  gc_ErrTranslation_fr_Text612 : WSTRING(60) := " [PIN_180 ]: EvPropGenerator -  Deviation of current control";
  gc_ErrTranslation_fr_Text613 : WSTRING(77) := " [PIN_180 ]: EvPropGenerator -  Internal error ( software or hardware error )";
  gc_ErrTranslation_fr_Text614 : WSTRING(65) := " [PIN_189 ]: EvServiceBrakeAxleOscillant -  Internal Driver Error";
  gc_ErrTranslation_fr_Text615 : WSTRING(13) := "Unknown error";
  gc_ErrTranslation_fr_Text616 : WSTRING(32) := "Short to Power has been detected";
  gc_ErrTranslation_fr_Text617 : WSTRING(33) := "Short to Ground has been detected";
  gc_ErrTranslation_fr_Text618 : WSTRING(15) := "Wrong Parameter";
  gc_ErrTranslation_fr_Text619 : WSTRING(13) := "Unknown error";
  gc_ErrTranslation_fr_Text620 : WSTRING(32) := "Short to Power has been detected";
  gc_ErrTranslation_fr_Text621 : WSTRING(33) := "Short to Ground has been detected";
  gc_ErrTranslation_fr_Text622 : WSTRING(15) := "Wrong Parameter";
  gc_ErrTranslation_fr_Text623 : WSTRING(13) := "Unknown error";
  gc_ErrTranslation_fr_Text624 : WSTRING(71) := " [PIN_193 ]: EvUpAxleOscillant -  HS OpenLoad / Short To Power external";
  gc_ErrTranslation_fr_Text625 : WSTRING(60) := " [PIN_193 ]: EvUpAxleOscillant -  HS Short To Power internal";
  gc_ErrTranslation_fr_Text626 : WSTRING(52) := " [PIN_193 ]: EvUpAxleOscillant -  HS Short To Ground";
  gc_ErrTranslation_fr_Text627 : WSTRING(55) := " [PIN_193 ]: EvUpAxleOscillant -  Internal Driver Error";
  gc_ErrTranslation_fr_Text628 : WSTRING(37) := "HS OpenLoad / Short To Power external";
  gc_ErrTranslation_fr_Text629 : WSTRING(26) := "HS Short To Power internal";
  gc_ErrTranslation_fr_Text630 : WSTRING(18) := "HS Short To Ground";
  gc_ErrTranslation_fr_Text631 : WSTRING(21) := "Internal Driver Error";
  gc_ErrTranslation_fr_Text632 : WSTRING(37) := "HS OpenLoad / Short To Power external";
  gc_ErrTranslation_fr_Text633 : WSTRING(26) := "HS Short To Power internal";
  gc_ErrTranslation_fr_Text634 : WSTRING(18) := "HS Short To Ground";
  gc_ErrTranslation_fr_Text635 : WSTRING(21) := "Internal Driver Error";
  gc_ErrTranslation_fr_Text636 : WSTRING(52) := "An input signal is too low / Short circuit to ground";
  gc_ErrTranslation_fr_Text637 : WSTRING(52) := "An input signal is too high / Short circuit to power";
  gc_ErrTranslation_fr_Text638 : WSTRING(37) := "An input signal is out of valid range";
  gc_ErrTranslation_fr_Text639 : WSTRING(39) := "Warning: a block has limited parameters";
  gc_ErrTranslation_fr_Text640 : WSTRING(23) := "An initialization error";
  gc_ErrTranslation_fr_Text641 : WSTRING(52) := "An input signal is too low / Short circuit to ground";
  gc_ErrTranslation_fr_Text642 : WSTRING(52) := "An input signal is too high / Short circuit to power";
  gc_ErrTranslation_fr_Text643 : WSTRING(37) := "An input signal is out of valid range";
  gc_ErrTranslation_fr_Text644 : WSTRING(39) := "Warning: a block has limited parameters";
  gc_ErrTranslation_fr_Text645 : WSTRING(23) := "An initialization error";
  gc_ErrTranslation_fr_Text646 : WSTRING(66) := " [PIN_196 ]: EvUpAxleFixe -  HS OpenLoad / Short To Power external";
  gc_ErrTranslation_fr_Text647 : WSTRING(55) := " [PIN_196 ]: EvUpAxleFixe -  HS Short To Power internal";
  gc_ErrTranslation_fr_Text648 : WSTRING(47) := " [PIN_196 ]: EvUpAxleFixe -  HS Short To Ground";
  gc_ErrTranslation_fr_Text649 : WSTRING(50) := " [PIN_196 ]: EvUpAxleFixe -  Internal Driver Error";
  gc_ErrTranslation_fr_Text650 : WSTRING(73) := " [PIN_169 ]: EvDownAxleOscillant -  HS OpenLoad / Short To Power external";
  gc_ErrTranslation_fr_Text651 : WSTRING(62) := " [PIN_149 ]: BlueFire -  HS OpenLoad / Short To Power external";
  gc_ErrTranslation_fr_Text652 : WSTRING(51) := " [PIN_149 ]: BlueFire -  HS Short To Power internal";
  gc_ErrTranslation_fr_Text653 : WSTRING(43) := " [PIN_149 ]: BlueFire -  HS Short To Ground";
  gc_ErrTranslation_fr_Text654 : WSTRING(46) := " [PIN_149 ]: BlueFire -  Internal Driver Error";
  gc_ErrTranslation_fr_Text655 : WSTRING(73) := " [PIN_173 ]: OrangeFlashingLight -  HS OpenLoad / Short To Power external";
  gc_ErrTranslation_fr_Text656 : WSTRING(62) := " [PIN_173 ]: OrangeFlashingLight -  HS Short To Power internal";
  gc_ErrTranslation_fr_Text657 : WSTRING(54) := " [PIN_173 ]: OrangeFlashingLight -  HS Short To Ground";
  gc_ErrTranslation_fr_Text658 : WSTRING(57) := " [PIN_173 ]: OrangeFlashingLight -  Internal Driver Error";
  gc_ErrTranslation_fr_Text659 : WSTRING(62) := " [PIN_169 ]: EvDownAxleOscillant -  HS Short To Power internal";
  gc_ErrTranslation_fr_Text660 : WSTRING(54) := " [PIN_169 ]: EvDownAxleOscillant -  HS Short To Ground";
  gc_ErrTranslation_fr_Text661 : WSTRING(57) := " [PIN_169 ]: EvDownAxleOscillant -  Internal Driver Error";
  gc_ErrTranslation_fr_Text662 : WSTRING(68) := " [PIN_172 ]: EvDownAxleFixe -  HS OpenLoad / Short To Power external";
  gc_ErrTranslation_fr_Text663 : WSTRING(62) := " [PIN_182 ]: EvBypass -  HS OpenLoad / Short To Power external";
  gc_ErrTranslation_fr_Text664 : WSTRING(51) := " [PIN_182 ]: EvBypass -  HS Short To Power internal";
  gc_ErrTranslation_fr_Text665 : WSTRING(43) := " [PIN_182 ]: EvBypass -  HS Short To Ground";
  gc_ErrTranslation_fr_Text666 : WSTRING(46) := " [PIN_182 ]: EvBypass -  Internal Driver Error";
  gc_ErrTranslation_fr_Text667 : WSTRING(57) := " [PIN_172 ]: EvDownAxleFixe -  HS Short To Power internal";
  gc_ErrTranslation_fr_Text668 : WSTRING(49) := " [PIN_172 ]: EvDownAxleFixe -  HS Short To Ground";
  gc_ErrTranslation_fr_Text669 : WSTRING(52) := " [PIN_172 ]: EvDownAxleFixe -  Internal Driver Error";
  gc_ErrTranslation_fr_Text670 : WSTRING(71) := " [PIN_191 ]: SupplyPvgDeltaArm -  HS OpenLoad / Short To Power external";
  gc_ErrTranslation_fr_Text671 : WSTRING(60) := " [PIN_191 ]: SupplyPvgDeltaArm -  HS Short To Power internal";
  gc_ErrTranslation_fr_Text672 : WSTRING(52) := " [PIN_191 ]: SupplyPvgDeltaArm -  HS Short To Ground";
  gc_ErrTranslation_fr_Text673 : WSTRING(55) := " [PIN_191 ]: SupplyPvgDeltaArm -  Internal Driver Error";
  gc_ErrTranslation_fr_Text674 : WSTRING(70) := " [PIN_167 ]: SupplyPvgBoomArm -  HS OpenLoad / Short To Power external";
  gc_ErrTranslation_fr_Text675 : WSTRING(59) := " [PIN_167 ]: SupplyPvgBoomArm -  HS Short To Power internal";
  gc_ErrTranslation_fr_Text676 : WSTRING(51) := " [PIN_167 ]: SupplyPvgBoomArm -  HS Short To Ground";
  gc_ErrTranslation_fr_Text677 : WSTRING(54) := " [PIN_167 ]: SupplyPvgBoomArm -  Internal Driver Error";
  gc_ErrTranslation_fr_Text678 : WSTRING(75) := " [PIN_194 ]: SupplyPvgTelescopeArm -  HS OpenLoad / Short To Power external";
  gc_ErrTranslation_fr_Text679 : WSTRING(64) := " [PIN_194 ]: SupplyPvgTelescopeArm -  HS Short To Power internal";
  gc_ErrTranslation_fr_Text680 : WSTRING(56) := " [PIN_194 ]: SupplyPvgTelescopeArm -  HS Short To Ground";
  gc_ErrTranslation_fr_Text681 : WSTRING(59) := " [PIN_194 ]: SupplyPvgTelescopeArm -  Internal Driver Error";
  gc_ErrTranslation_fr_Text682 : WSTRING(72) := " [PIN_170 ]: SupplyPvgPropEvTOR -  HS OpenLoad / Short To Power external";
  gc_ErrTranslation_fr_Text683 : WSTRING(61) := " [PIN_170 ]: SupplyPvgPropEvTOR -  HS Short To Power internal";
  gc_ErrTranslation_fr_Text684 : WSTRING(53) := " [PIN_170 ]: SupplyPvgPropEvTOR -  HS Short To Ground";
  gc_ErrTranslation_fr_Text685 : WSTRING(56) := " [PIN_170 ]: SupplyPvgPropEvTOR -  Internal Driver Error";
  gc_ErrTranslation_fr_Text686 : WSTRING(83) := " [PIN_110 ]: RailHookSensor -  An input signal is too high / Short circuit to power";
  gc_ErrTranslation_fr_Text687 : WSTRING(68) := " [PIN_110 ]: RailHookSensor -  An input signal is out of valid range";
  gc_ErrTranslation_fr_Text688 : WSTRING(70) := " [PIN_110 ]: RailHookSensor -  Warning: a block has limited parameters";
  gc_ErrTranslation_fr_Text689 : WSTRING(54) := " [PIN_110 ]: RailHookSensor -  An initialization error";
  gc_ErrTranslation_fr_Text690 : WSTRING(88) := " [PIN_134 ]: InductiveRailSensor -  An input signal is too low / Short circuit to ground";
  gc_ErrTranslation_fr_Text691 : WSTRING(88) := " [PIN_134 ]: InductiveRailSensor -  An input signal is too high / Short circuit to power";
  gc_ErrTranslation_fr_Text692 : WSTRING(73) := " [PIN_134 ]: InductiveRailSensor -  An input signal is out of valid range";
  gc_ErrTranslation_fr_Text693 : WSTRING(75) := " [PIN_134 ]: InductiveRailSensor -  Warning: a block has limited parameters";
  gc_ErrTranslation_fr_Text694 : WSTRING(59) := " [PIN_134 ]: InductiveRailSensor -  An initialization error";
  gc_ErrTranslation_fr_Text695 : WSTRING(83) := " [PIN_111 ]: CenteredTurret -  An input signal is too low / Short circuit to ground";
  gc_ErrTranslation_fr_Text696 : WSTRING(83) := " [PIN_111 ]: CenteredTurret -  An input signal is too high / Short circuit to power";
  gc_ErrTranslation_fr_Text697 : WSTRING(68) := " [PIN_111 ]: CenteredTurret -  An input signal is out of valid range";
  gc_ErrTranslation_fr_Text698 : WSTRING(70) := " [PIN_111 ]: CenteredTurret -  Warning: a block has limited parameters";
  gc_ErrTranslation_fr_Text699 : WSTRING(54) := " [PIN_111 ]: CenteredTurret -  An initialization error";
  gc_ErrTranslation_fr_Text700 : WSTRING(85) := " [PIN_135 ]: WorkKeyTrackSide -  An input signal is too low / Short circuit to ground";
  gc_ErrTranslation_fr_Text701 : WSTRING(85) := " [PIN_135 ]: WorkKeyTrackSide -  An input signal is too high / Short circuit to power";
  gc_ErrTranslation_fr_Text702 : WSTRING(70) := " [PIN_135 ]: WorkKeyTrackSide -  An input signal is out of valid range";
  gc_ErrTranslation_fr_Text703 : WSTRING(72) := " [PIN_135 ]: WorkKeyTrackSide -  Warning: a block has limited parameters";
  gc_ErrTranslation_fr_Text704 : WSTRING(56) := " [PIN_135 ]: WorkKeyTrackSide -  An initialization error";
  gc_ErrTranslation_fr_Text705 : WSTRING(85) := " [PIN_136 ]: WorkKeyBilateral -  An input signal is too low / Short circuit to ground";
  gc_ErrTranslation_fr_Text706 : WSTRING(85) := " [PIN_136 ]: WorkKeyBilateral -  An input signal is too high / Short circuit to power";
  gc_ErrTranslation_fr_Text707 : WSTRING(70) := " [PIN_136 ]: WorkKeyBilateral -  An input signal is out of valid range";
  gc_ErrTranslation_fr_Text708 : WSTRING(72) := " [PIN_136 ]: WorkKeyBilateral -  Warning: a block has limited parameters";
  gc_ErrTranslation_fr_Text709 : WSTRING(56) := " [PIN_136 ]: WorkKeyBilateral -  An initialization error";
  gc_ErrTranslation_fr_Text710 : WSTRING(83) := " [PIN_113 ]: WorkKeyCentred -  An input signal is too low / Short circuit to ground";
  gc_ErrTranslation_fr_Text711 : WSTRING(83) := " [PIN_113 ]: WorkKeyCentred -  An input signal is too high / Short circuit to power";
  gc_ErrTranslation_fr_Text712 : WSTRING(68) := " [PIN_113 ]: WorkKeyCentred -  An input signal is out of valid range";
  gc_ErrTranslation_fr_Text713 : WSTRING(70) := " [PIN_113 ]: WorkKeyCentred -  Warning: a block has limited parameters";
  gc_ErrTranslation_fr_Text714 : WSTRING(54) := " [PIN_113 ]: WorkKeyCentred -  An initialization error";
  gc_ErrTranslation_fr_Text715 : WSTRING(92) := " [PIN_137 ]: AbutmentTurretTrackSide -  An input signal is too low / Short circuit to ground";
  gc_ErrTranslation_fr_Text716 : WSTRING(92) := " [PIN_137 ]: AbutmentTurretTrackSide -  An input signal is too high / Short circuit to power";
  gc_ErrTranslation_fr_Text717 : WSTRING(77) := " [PIN_137 ]: AbutmentTurretTrackSide -  An input signal is out of valid range";
  gc_ErrTranslation_fr_Text718 : WSTRING(79) := " [PIN_137 ]: AbutmentTurretTrackSide -  Warning: a block has limited parameters";
  gc_ErrTranslation_fr_Text719 : WSTRING(63) := " [PIN_137 ]: AbutmentTurretTrackSide -  An initialization error";
  gc_ErrTranslation_fr_Text720 : WSTRING(94) := " [PIN_138 ]: AbutmentTurretCentredSide -  An input signal is too low / Short circuit to ground";
  gc_ErrTranslation_fr_Text721 : WSTRING(94) := " [PIN_138 ]: AbutmentTurretCentredSide -  An input signal is too high / Short circuit to power";
  gc_ErrTranslation_fr_Text722 : WSTRING(79) := " [PIN_138 ]: AbutmentTurretCentredSide -  An input signal is out of valid range";
  gc_ErrTranslation_fr_Text723 : WSTRING(81) := " [PIN_138 ]: AbutmentTurretCentredSide -  Warning: a block has limited parameters";
  gc_ErrTranslation_fr_Text724 : WSTRING(65) := " [PIN_138 ]: AbutmentTurretCentredSide -  An initialization error";
  gc_ErrTranslation_fr_Text725 : WSTRING(96) := " [PIN_139 ]: OscillantAxleSpeedSensorDir -  An input signal is too low / Short circuit to ground";
  gc_ErrTranslation_fr_Text726 : WSTRING(96) := " [PIN_139 ]: OscillantAxleSpeedSensorDir -  An input signal is too high / Short circuit to power";
  gc_ErrTranslation_fr_Text727 : WSTRING(81) := " [PIN_139 ]: OscillantAxleSpeedSensorDir -  An input signal is out of valid range";
  gc_ErrTranslation_fr_Text728 : WSTRING(83) := " [PIN_139 ]: OscillantAxleSpeedSensorDir -  Warning: a block has limited parameters";
  gc_ErrTranslation_fr_Text729 : WSTRING(67) := " [PIN_139 ]: OscillantAxleSpeedSensorDir -  An initialization error";
  gc_ErrTranslation_fr_Text730 : WSTRING(91) := " [PIN_140 ]: FixeAxleSpeedSensorDir -  An input signal is too low / Short circuit to ground";
  gc_ErrTranslation_fr_Text731 : WSTRING(91) := " [PIN_140 ]: FixeAxleSpeedSensorDir -  An input signal is too high / Short circuit to power";
  gc_ErrTranslation_fr_Text732 : WSTRING(76) := " [PIN_140 ]: FixeAxleSpeedSensorDir -  An input signal is out of valid range";
  gc_ErrTranslation_fr_Text733 : WSTRING(78) := " [PIN_140 ]: FixeAxleSpeedSensorDir -  Warning: a block has limited parameters";
  gc_ErrTranslation_fr_Text734 : WSTRING(62) := " [PIN_140 ]: FixeAxleSpeedSensorDir -  An initialization error";
  gc_ErrTranslation_fr_Text735 : WSTRING(81) := " [PIN_117 ]: TrailerGache -  An input signal is too low / Short circuit to ground";
  gc_ErrTranslation_fr_Text736 : WSTRING(81) := " [PIN_117 ]: TrailerGache -  An input signal is too high / Short circuit to power";
  gc_ErrTranslation_fr_Text737 : WSTRING(66) := " [PIN_117 ]: TrailerGache -  An input signal is out of valid range";
  gc_ErrTranslation_fr_Text738 : WSTRING(68) := " [PIN_117 ]: TrailerGache -  Warning: a block has limited parameters";
  gc_ErrTranslation_fr_Text739 : WSTRING(52) := " [PIN_117 ]: TrailerGache -  An initialization error";
  gc_ErrTranslation_fr_Text740 : WSTRING(94) := " [PIN_141 ]: MeasuringMastSensorFolded -  An input signal is too low / Short circuit to ground";
  gc_ErrTranslation_fr_Text741 : WSTRING(94) := " [PIN_141 ]: MeasuringMastSensorFolded -  An input signal is too high / Short circuit to power";
  gc_ErrTranslation_fr_Text742 : WSTRING(79) := " [PIN_141 ]: MeasuringMastSensorFolded -  An input signal is out of valid range";
  gc_ErrTranslation_fr_Text743 : WSTRING(81) := " [PIN_141 ]: MeasuringMastSensorFolded -  Warning: a block has limited parameters";
  gc_ErrTranslation_fr_Text744 : WSTRING(65) := " [PIN_141 ]: MeasuringMastSensorFolded -  An initialization error";
  gc_ErrTranslation_fr_Text745 : WSTRING(80) := " [PIN_124 ]: Aru1Contact -  An input signal is too low / Short circuit to ground";
  gc_ErrTranslation_fr_Text746 : WSTRING(80) := " [PIN_124 ]: Aru1Contact -  An input signal is too high / Short circuit to power";
  gc_ErrTranslation_fr_Text747 : WSTRING(65) := " [PIN_124 ]: Aru1Contact -  An input signal is out of valid range";
  gc_ErrTranslation_fr_Text748 : WSTRING(67) := " [PIN_124 ]: Aru1Contact -  Warning: a block has limited parameters";
  gc_ErrTranslation_fr_Text749 : WSTRING(54) := " [PIN_101 ]: EvForwardPump -  Open load / open circuit";
  gc_ErrTranslation_fr_Text750 : WSTRING(69) := " [PIN_101 ]: EvForwardPump -  Short circuit to power supply / battery";
  gc_ErrTranslation_fr_Text751 : WSTRING(53) := " [PIN_101 ]: EvForwardPump -  Short circuit to ground";
  gc_ErrTranslation_fr_Text752 : WSTRING(58) := " [PIN_101 ]: EvForwardPump -  Deviation of current control";
  gc_ErrTranslation_fr_Text753 : WSTRING(75) := " [PIN_101 ]: EvForwardPump -  Internal error ( software or hardware error )";
  gc_ErrTranslation_fr_Text754 : WSTRING(55) := " [PIN_125 ]: EvBackwardPump -  Open load / open circuit";
  gc_ErrTranslation_fr_Text755 : WSTRING(70) := " [PIN_125 ]: EvBackwardPump -  Short circuit to power supply / battery";
  gc_ErrTranslation_fr_Text756 : WSTRING(54) := " [PIN_125 ]: EvBackwardPump -  Short circuit to ground";
  gc_ErrTranslation_fr_Text757 : WSTRING(59) := " [PIN_125 ]: EvBackwardPump -  Deviation of current control";
  gc_ErrTranslation_fr_Text758 : WSTRING(76) := " [PIN_125 ]: EvBackwardPump -  Internal error ( software or hardware error )";
  gc_ErrTranslation_fr_Text759 : WSTRING(72) := " [PIN_194 ]: WhiteTrailerLights -  HS OpenLoad / Short To Power external";
  gc_ErrTranslation_fr_Text760 : WSTRING(61) := " [PIN_194 ]: WhiteTrailerLights -  HS Short To Power internal";
  gc_ErrTranslation_fr_Text761 : WSTRING(53) := " [PIN_194 ]: WhiteTrailerLights -  HS Short To Ground";
  gc_ErrTranslation_fr_Text762 : WSTRING(56) := " [PIN_194 ]: WhiteTrailerLights -  Internal Driver Error";
  gc_ErrTranslation_fr_Text763 : WSTRING(70) := " [PIN_170 ]: RedTrailerLights -  HS OpenLoad / Short To Power external";
  gc_ErrTranslation_fr_Text764 : WSTRING(59) := " [PIN_170 ]: RedTrailerLights -  HS Short To Power internal";
  gc_ErrTranslation_fr_Text765 : WSTRING(51) := " [PIN_170 ]: RedTrailerLights -  HS Short To Ground";
  gc_ErrTranslation_fr_Text766 : WSTRING(54) := " [PIN_170 ]: RedTrailerLights -  Internal Driver Error";
  gc_ErrTranslation_fr_Text767 : WSTRING(87) := " [PIN_131 ]: TurretPostSelector -  An input signal is too low / Short circuit to ground";
  gc_ErrTranslation_fr_Text768 : WSTRING(87) := " [PIN_131 ]: TurretPostSelector -  An input signal is too high / Short circuit to power";
  gc_ErrTranslation_fr_Text769 : WSTRING(72) := " [PIN_131 ]: TurretPostSelector -  An input signal is out of valid range";
  gc_ErrTranslation_fr_Text770 : WSTRING(74) := " [PIN_131 ]: TurretPostSelector -  Warning: a block has limited parameters";
  gc_ErrTranslation_fr_Text771 : WSTRING(58) := " [PIN_131 ]: TurretPostSelector -  An initialization error";
  gc_ErrTranslation_fr_Text772 : WSTRING(86) := " [PIN_108 ]: RadioPostSelector -  An input signal is too low / Short circuit to ground";
  gc_ErrTranslation_fr_Text773 : WSTRING(86) := " [PIN_108 ]: RadioPostSelector -  An input signal is too high / Short circuit to power";
  gc_ErrTranslation_fr_Text774 : WSTRING(71) := " [PIN_108 ]: RadioPostSelector -  An input signal is out of valid range";
  gc_ErrTranslation_fr_Text775 : WSTRING(73) := " [PIN_108 ]: RadioPostSelector -  Warning: a block has limited parameters";
  gc_ErrTranslation_fr_Text776 : WSTRING(57) := " [PIN_108 ]: RadioPostSelector -  An initialization error";
  gc_ErrTranslation_fr_Text777 : WSTRING(88) := " [PIN_132 ]: NacellePostSelector -  An input signal is too low / Short circuit to ground";
  gc_ErrTranslation_fr_Text778 : WSTRING(88) := " [PIN_132 ]: NacellePostSelector -  An input signal is too high / Short circuit to power";
  gc_ErrTranslation_fr_Text779 : WSTRING(73) := " [PIN_132 ]: NacellePostSelector -  An input signal is out of valid range";
  gc_ErrTranslation_fr_Text780 : WSTRING(75) := " [PIN_132 ]: NacellePostSelector -  Warning: a block has limited parameters";
  gc_ErrTranslation_fr_Text781 : WSTRING(59) := " [PIN_132 ]: NacellePostSelector -  An initialization error";
  gc_ErrTranslation_fr_Text782 : WSTRING(89) := " [PIN_117 ]: DeltaArmFoldedSensor -  An input signal is too low / Short circuit to ground";
  gc_ErrTranslation_fr_Text783 : WSTRING(89) := " [PIN_117 ]: DeltaArmFoldedSensor -  An input signal is too high / Short circuit to power";
  gc_ErrTranslation_fr_Text784 : WSTRING(74) := " [PIN_117 ]: DeltaArmFoldedSensor -  An input signal is out of valid range";
  gc_ErrTranslation_fr_Text785 : WSTRING(76) := " [PIN_117 ]: DeltaArmFoldedSensor -  Warning: a block has limited parameters";
  gc_ErrTranslation_fr_Text786 : WSTRING(60) := " [PIN_117 ]: DeltaArmFoldedSensor -  An initialization error";
  gc_ErrTranslation_fr_Text787 : WSTRING(88) := " [PIN_141 ]: BoomArmFoldedSensor -  An input signal is too low / Short circuit to ground";
  gc_ErrTranslation_fr_Text788 : WSTRING(88) := " [PIN_141 ]: BoomArmFoldedSensor -  An input signal is too high / Short circuit to power";
  gc_ErrTranslation_fr_Text789 : WSTRING(73) := " [PIN_141 ]: BoomArmFoldedSensor -  An input signal is out of valid range";
  gc_ErrTranslation_fr_Text790 : WSTRING(75) := " [PIN_141 ]: BoomArmFoldedSensor -  Warning: a block has limited parameters";
  gc_ErrTranslation_fr_Text791 : WSTRING(59) := " [PIN_141 ]: BoomArmFoldedSensor -  An initialization error";
  gc_ErrTranslation_fr_Text792 : WSTRING(87) := " [PIN_148 ]: AlternatorChargeOK -  An input signal is too low / Short circuit to ground";
  gc_ErrTranslation_fr_Text793 : WSTRING(87) := " [PIN_148 ]: AlternatorChargeOK -  An input signal is too high / Short circuit to power";
  gc_ErrTranslation_fr_Text794 : WSTRING(72) := " [PIN_148 ]: AlternatorChargeOK -  An input signal is out of valid range";
  gc_ErrTranslation_fr_Text795 : WSTRING(74) := " [PIN_148 ]: AlternatorChargeOK -  Warning: a block has limited parameters";
  gc_ErrTranslation_fr_Text796 : WSTRING(58) := " [PIN_148 ]: AlternatorChargeOK -  An initialization error";
  gc_ErrTranslation_fr_Text797 : WSTRING(70) := " [PIN_176 ]: OverloadSecurity -  HS OpenLoad / Short To Power external";
  gc_ErrTranslation_fr_Text798 : WSTRING(59) := " [PIN_176 ]: OverloadSecurity -  HS Short To Power internal";
  gc_ErrTranslation_fr_Text799 : WSTRING(51) := " [PIN_176 ]: OverloadSecurity -  HS Short To Ground";
  gc_ErrTranslation_fr_Text800 : WSTRING(54) := " [PIN_176 ]: OverloadSecurity -  Internal Driver Error";
  gc_ErrTranslation_fr_Text801 : WSTRING(70) := " [PIN_152 ]: SupllyTorSensors -  HS OpenLoad / Short To Power external";
  gc_ErrTranslation_fr_Text802 : WSTRING(59) := " [PIN_152 ]: SupllyTorSensors -  HS Short To Power internal";
  gc_ErrTranslation_fr_Text803 : WSTRING(51) := " [PIN_152 ]: SupllyTorSensors -  HS Short To Ground";
  gc_ErrTranslation_fr_Text804 : WSTRING(54) := " [PIN_152 ]: SupllyTorSensors -  Internal Driver Error";
  gc_ErrTranslation_fr_Text805 : WSTRING(51) := " [PIN_124 ]: Aru1Contact -  An initialization error";
  gc_ErrTranslation_fr_Text806 : WSTRING(80) := " [PIN_148 ]: Aru2Contact -  An input signal is too low / Short circuit to ground";
  gc_ErrTranslation_fr_Text807 : WSTRING(80) := " [PIN_148 ]: Aru2Contact -  An input signal is too high / Short circuit to power";
  gc_ErrTranslation_fr_Text808 : WSTRING(65) := " [PIN_148 ]: Aru2Contact -  An input signal is out of valid range";
  gc_ErrTranslation_fr_Text809 : WSTRING(70) := " [PIN_153 ]: SupllyAnaSensors -  HS OpenLoad / Short To Power external";
  gc_ErrTranslation_fr_Text810 : WSTRING(59) := " [PIN_153 ]: SupllyAnaSensors -  HS Short To Power internal";
  gc_ErrTranslation_fr_Text811 : WSTRING(51) := " [PIN_153 ]: SupllyAnaSensors -  HS Short To Ground";
  gc_ErrTranslation_fr_Text812 : WSTRING(54) := " [PIN_153 ]: SupllyAnaSensors -  Internal Driver Error";
  gc_ErrTranslation_fr_Text813 : WSTRING(68) := " [PIN_159 ]: EvSyncRotation -  HS OpenLoad / Short To Power external";
  gc_ErrTranslation_fr_Text814 : WSTRING(57) := " [PIN_159 ]: EvSyncRotation -  HS Short To Power internal";
  gc_ErrTranslation_fr_Text815 : WSTRING(49) := " [PIN_159 ]: EvSyncRotation -  HS Short To Ground";
  gc_ErrTranslation_fr_Text816 : WSTRING(52) := " [PIN_159 ]: EvSyncRotation -  Internal Driver Error";
  gc_ErrTranslation_fr_Text817 : WSTRING(70) := " [PIN_156 ]: SupplyAnaSensors -  HS OpenLoad / Short To Power external";
  gc_ErrTranslation_fr_Text818 : WSTRING(59) := " [PIN_156 ]: SupplyAnaSensors -  HS Short To Power internal";
  gc_ErrTranslation_fr_Text819 : WSTRING(51) := " [PIN_156 ]: SupplyAnaSensors -  HS Short To Ground";
  gc_ErrTranslation_fr_Text820 : WSTRING(54) := " [PIN_156 ]: SupplyAnaSensors -  Internal Driver Error";
  gc_ErrTranslation_fr_Text821 : WSTRING(67) := " [PIN_148 ]: Aru2Contact -  Warning: a block has limited parameters";
  gc_ErrTranslation_fr_Text822 : WSTRING(51) := " [PIN_148 ]: Aru2Contact -  An initialization error";
  gc_ErrTranslation_fr_Text823 : WSTRING(85) := " [PIN_128 ]: AruRadio1Contact -  An input signal is too low / Short circuit to ground";
  gc_ErrTranslation_fr_Text824 : WSTRING(85) := " [PIN_128 ]: AruRadio1Contact -  An input signal is too high / Short circuit to power";
  gc_ErrTranslation_fr_Text825 : WSTRING(70) := " [PIN_128 ]: AruRadio1Contact -  An input signal is out of valid range";
  gc_ErrTranslation_fr_Text826 : WSTRING(72) := " [PIN_128 ]: AruRadio1Contact -  Warning: a block has limited parameters";
  gc_ErrTranslation_fr_Text827 : WSTRING(56) := " [PIN_128 ]: AruRadio1Contact -  An initialization error";
  gc_ErrTranslation_fr_Text828 : WSTRING(85) := " [PIN_105 ]: AruRadio2Contact -  An input signal is too low / Short circuit to ground";
  gc_ErrTranslation_fr_Text829 : WSTRING(85) := " [PIN_105 ]: AruRadio2Contact -  An input signal is too high / Short circuit to power";
  gc_ErrTranslation_fr_Text830 : WSTRING(70) := " [PIN_105 ]: AruRadio2Contact -  An input signal is out of valid range";
  gc_ErrTranslation_fr_Text831 : WSTRING(72) := " [PIN_105 ]: AruRadio2Contact -  Warning: a block has limited parameters";
  gc_ErrTranslation_fr_Text832 : WSTRING(56) := " [PIN_105 ]: AruRadio2Contact -  An initialization error";
  gc_ErrTranslation_fr_Text833 : WSTRING(64) := " [PIN_183 ]: Noisemaker -  HS OpenLoad / Short To Power external";
  gc_ErrTranslation_fr_Text834 : WSTRING(53) := " [PIN_183 ]: Noisemaker -  HS Short To Power internal";
  gc_ErrTranslation_fr_Text835 : WSTRING(45) := " [PIN_183 ]: Noisemaker -  HS Short To Ground";
  gc_ErrTranslation_fr_Text836 : WSTRING(48) := " [PIN_183 ]: Noisemaker -  Internal Driver Error";
  gc_ErrTranslation_fr_Text837 : WSTRING(72) := " [PIN_154 ]: EvRotTurretClkwise -  HS OpenLoad / Short To Power external";
  gc_ErrTranslation_fr_Text838 : WSTRING(61) := " [PIN_154 ]: EvRotTurretClkwise -  HS Short To Power internal";
  gc_ErrTranslation_fr_Text839 : WSTRING(53) := " [PIN_154 ]: EvRotTurretClkwise -  HS Short To Ground";
  gc_ErrTranslation_fr_Text840 : WSTRING(56) := " [PIN_154 ]: EvRotTurretClkwise -  Internal Driver Error";
  gc_ErrTranslation_fr_Text841 : WSTRING(74) := " [PIN_178 ]: EvRotTurretCtClkwise -  HS OpenLoad / Short To Power external";
  gc_ErrTranslation_fr_Text842 : WSTRING(63) := " [PIN_178 ]: EvRotTurretCtClkwise -  HS Short To Power internal";
  gc_ErrTranslation_fr_Text843 : WSTRING(55) := " [PIN_178 ]: EvRotTurretCtClkwise -  HS Short To Ground";
  gc_ErrTranslation_fr_Text844 : WSTRING(58) := " [PIN_178 ]: EvRotTurretCtClkwise -  Internal Driver Error";
  gc_ErrTranslation_fr_Text845 : WSTRING(74) := " [PIN_157 ]: EvRotBasketCtClkwise -  HS OpenLoad / Short To Power external";
  gc_ErrTranslation_fr_Text846 : WSTRING(63) := " [PIN_157 ]: EvRotBasketCtClkwise -  HS Short To Power internal";
  gc_ErrTranslation_fr_Text847 : WSTRING(55) := " [PIN_157 ]: EvRotBasketCtClkwise -  HS Short To Ground";
  gc_ErrTranslation_fr_Text848 : WSTRING(58) := " [PIN_157 ]: EvRotBasketCtClkwise -  Internal Driver Error";
  gc_ErrTranslation_fr_Text849 : WSTRING(72) := " [PIN_181 ]: EvRotBasketClkwise -  HS OpenLoad / Short To Power external";
  gc_ErrTranslation_fr_Text850 : WSTRING(61) := " [PIN_181 ]: EvRotBasketClkwise -  HS Short To Power internal";
  gc_ErrTranslation_fr_Text851 : WSTRING(53) := " [PIN_181 ]: EvRotBasketClkwise -  HS Short To Ground";
  gc_ErrTranslation_fr_Text852 : WSTRING(56) := " [PIN_181 ]: EvRotBasketClkwise -  Internal Driver Error";
  gc_ErrTranslation_fr_Text853 : WSTRING(66) := " [PIN_160 ]: EvUpPendular -  HS OpenLoad / Short To Power external";
  gc_ErrTranslation_fr_Text854 : WSTRING(55) := " [PIN_160 ]: EvUpPendular -  HS Short To Power internal";
  gc_ErrTranslation_fr_Text855 : WSTRING(47) := " [PIN_160 ]: EvUpPendular -  HS Short To Ground";
  gc_ErrTranslation_fr_Text856 : WSTRING(50) := " [PIN_160 ]: EvUpPendular -  Internal Driver Error";
  gc_ErrTranslation_fr_Text857 : WSTRING(68) := " [PIN_184 ]: EvDownPendular -  HS OpenLoad / Short To Power external";
  gc_ErrTranslation_fr_Text858 : WSTRING(57) := " [PIN_184 ]: EvDownPendular -  HS Short To Power internal";
  gc_ErrTranslation_fr_Text859 : WSTRING(49) := " [PIN_184 ]: EvDownPendular -  HS Short To Ground";
  gc_ErrTranslation_fr_Text860 : WSTRING(52) := " [PIN_184 ]: EvDownPendular -  Internal Driver Error";
  gc_ErrTranslation_fr_Text861 : WSTRING(75) := " [PIN_187 ]: EvUpInclinaisonBasket -  HS OpenLoad / Short To Power external";
  gc_ErrTranslation_fr_Text862 : WSTRING(64) := " [PIN_187 ]: EvUpInclinaisonBasket -  HS Short To Power internal";
  gc_ErrTranslation_fr_Text863 : WSTRING(56) := " [PIN_187 ]: EvUpInclinaisonBasket -  HS Short To Ground";
  gc_ErrTranslation_fr_Text864 : WSTRING(59) := " [PIN_187 ]: EvUpInclinaisonBasket -  Internal Driver Error";
  gc_ErrTranslation_fr_Text865 : WSTRING(77) := " [PIN_163 ]: EvDownInclinaisonBasket -  HS OpenLoad / Short To Power external";
  gc_ErrTranslation_fr_Text866 : WSTRING(66) := " [PIN_163 ]: EvDownInclinaisonBasket -  HS Short To Power internal";
  gc_ErrTranslation_fr_Text867 : WSTRING(58) := " [PIN_163 ]: EvDownInclinaisonBasket -  HS Short To Ground";
  gc_ErrTranslation_fr_Text868 : WSTRING(61) := " [PIN_163 ]: EvDownInclinaisonBasket -  Internal Driver Error";
  gc_ErrTranslation_fr_Text869 : WSTRING(73) := " [PIN_137 ]: Aru1 -  An input signal is too low / Short circuit to ground";
  gc_ErrTranslation_fr_Text870 : WSTRING(73) := " [PIN_137 ]: Aru1 -  An input signal is too high / Short circuit to power";
  gc_ErrTranslation_fr_Text871 : WSTRING(58) := " [PIN_137 ]: Aru1 -  An input signal is out of valid range";
  gc_ErrTranslation_fr_Text872 : WSTRING(60) := " [PIN_137 ]: Aru1 -  Warning: a block has limited parameters";
  gc_ErrTranslation_fr_Text873 : WSTRING(44) := " [PIN_137 ]: Aru1 -  An initialization error";
  gc_ErrTranslation_fr_Text874 : WSTRING(73) := " [PIN_138 ]: Aru2 -  An input signal is too low / Short circuit to ground";
  gc_ErrTranslation_fr_Text875 : WSTRING(73) := " [PIN_138 ]: Aru2 -  An input signal is too high / Short circuit to power";
  gc_ErrTranslation_fr_Text876 : WSTRING(58) := " [PIN_138 ]: Aru2 -  An input signal is out of valid range";
  gc_ErrTranslation_fr_Text877 : WSTRING(60) := " [PIN_138 ]: Aru2 -  Warning: a block has limited parameters";
  gc_ErrTranslation_fr_Text878 : WSTRING(44) := " [PIN_138 ]: Aru2 -  An initialization error";
  gc_ErrTranslation_fr_Text879 : WSTRING(92) := " [PIN_113 ]: EntryTelescopeFdcSensor -  An input signal is too low / Short circuit to ground";
  gc_ErrTranslation_fr_Text880 : WSTRING(92) := " [PIN_113 ]: EntryTelescopeFdcSensor -  An input signal is too high / Short circuit to power";
  gc_ErrTranslation_fr_Text881 : WSTRING(77) := " [PIN_113 ]: EntryTelescopeFdcSensor -  An input signal is out of valid range";
  gc_ErrTranslation_fr_Text882 : WSTRING(79) := " [PIN_113 ]: EntryTelescopeFdcSensor -  Warning: a block has limited parameters";
  gc_ErrTranslation_fr_Text883 : WSTRING(63) := " [PIN_113 ]: EntryTelescopeFdcSensor -  An initialization error";
  gc_ErrTranslation_fr_Text884 : WSTRING(76) := " [PIN_165 ]: EvServiceBrakeAxleFixe -  HS OpenLoad / Short To Power external";
  gc_ErrTranslation_fr_Text885 : WSTRING(65) := " [PIN_165 ]: EvServiceBrakeAxleFixe -  HS Short To Power internal";
  gc_ErrTranslation_fr_Text886 : WSTRING(57) := " [PIN_165 ]: EvServiceBrakeAxleFixe -  HS Short To Ground";
  gc_ErrTranslation_fr_Text887 : WSTRING(60) := " [PIN_165 ]: EvServiceBrakeAxleFixe -  Internal Driver Error";
  gc_ErrTranslation_fr_Text888 : WSTRING(65) := " [-]: SpecificErrorC0 -  if Aru contact is pushed , stop movement";
  gc_ErrTranslation_fr_Text889 : WSTRING(63) := " [-]: SpecificErrorC0 -  if Aru radio is pushed , stop movement";
  gc_ErrTranslation_fr_Text890 : WSTRING(65) := " [-]: SpecificErrorC1 -  if Aru contact is pushed , stop movement";
  gc_ErrTranslation_fr_Text891 : WSTRING(63) := " [-]: SpecificErrorC1 -  if Aru radio is pushed , stop movement";
  gc_ErrTranslation_fr_Text892 : WSTRING(81) := " [PIN_252 ]: ReturnLowSideEvProGenerator -  HS OpenLoad / Short To Power external";
  gc_ErrTranslation_fr_Text893 : WSTRING(70) := " [PIN_252 ]: ReturnLowSideEvProGenerator -  HS Short To Power internal";
  gc_ErrTranslation_fr_Text894 : WSTRING(62) := " [PIN_252 ]: ReturnLowSideEvProGenerator -  HS Short To Ground";
  gc_ErrTranslation_fr_Text895 : WSTRING(65) := " [PIN_252 ]: ReturnLowSideEvProGenerator -  Internal Driver Error";
  gc_ErrTranslation_fr_Text896 : WSTRING(80) := " [PIN_104 PIN_128 ]: DeltaArmAngularSensor -  Master input signal short to power";
  gc_ErrTranslation_fr_Text897 : WSTRING(81) := " [PIN_104 PIN_128 ]: DeltaArmAngularSensor -  Master input signal short to ground";
  gc_ErrTranslation_fr_Text898 : WSTRING(79) := " [PIN_104 PIN_128 ]: DeltaArmAngularSensor -  Slave input signal short to power";
  gc_ErrTranslation_fr_Text899 : WSTRING(80) := " [PIN_104 PIN_128 ]: DeltaArmAngularSensor -  Slave input signal short to ground";
  gc_ErrTranslation_fr_Text900 : WSTRING(79) := " [PIN_104 PIN_128 ]: DeltaArmAngularSensor -  Deviation of signals out of limit";
  gc_ErrTranslation_fr_Text901 : WSTRING(62) := " [PIN_104 PIN_128 ]: DeltaArmAngularSensor -  Limp mode active";
  gc_ErrTranslation_fr_Text902 : WSTRING(81) := " [PIN_104 PIN_128 ]: DeltaArmAngularSensor -  Parameter of input char NOT monoton";
  gc_ErrTranslation_fr_Text903 : WSTRING(68) := " [PIN_104 PIN_128 ]: DeltaArmAngularSensor -  Unknown internal error";
  gc_ErrTranslation_fr_Text904 : WSTRING(80) := " [PIN_105 PIN_129 ]: ArrowArmAngularSensor -  Master input signal short to power";
  gc_ErrTranslation_fr_Text905 : WSTRING(81) := " [PIN_105 PIN_129 ]: ArrowArmAngularSensor -  Master input signal short to ground";
  gc_ErrTranslation_fr_Text906 : WSTRING(79) := " [PIN_105 PIN_129 ]: ArrowArmAngularSensor -  Slave input signal short to power";
  gc_ErrTranslation_fr_Text907 : WSTRING(80) := " [PIN_105 PIN_129 ]: ArrowArmAngularSensor -  Slave input signal short to ground";
  gc_ErrTranslation_fr_Text908 : WSTRING(79) := " [PIN_105 PIN_129 ]: ArrowArmAngularSensor -  Deviation of signals out of limit";
  gc_ErrTranslation_fr_Text909 : WSTRING(62) := " [PIN_105 PIN_129 ]: ArrowArmAngularSensor -  Limp mode active";
  gc_ErrTranslation_fr_Text910 : WSTRING(81) := " [PIN_105 PIN_129 ]: ArrowArmAngularSensor -  Parameter of input char NOT monoton";
  gc_ErrTranslation_fr_Text911 : WSTRING(68) := " [PIN_105 PIN_129 ]: ArrowArmAngularSensor -  Unknown internal error";
  gc_ErrTranslation_fr_Text912 : WSTRING(82) := " [-]: SpecificErrorC1 -  if stop all movement is detect by limit envelope function";
  gc_ErrTranslation_fr_Text913 : WSTRING(64) := " [PIN_154 ]: NeonLights -  HS OpenLoad / Short To Power external";
  gc_ErrTranslation_fr_Text914 : WSTRING(53) := " [PIN_154 ]: NeonLights -  HS Short To Power internal";
  gc_ErrTranslation_fr_Text915 : WSTRING(45) := " [PIN_154 ]: NeonLights -  HS Short To Ground";
  gc_ErrTranslation_fr_Text916 : WSTRING(48) := " [PIN_154 ]: NeonLights -  Internal Driver Error";
  gc_ErrTranslation_fr_Text917 : WSTRING(78) := " [PIN_159 ]: Ev2DeflectorTransmission -  HS OpenLoad / Short To Power external";
  gc_ErrTranslation_fr_Text918 : WSTRING(67) := " [PIN_159 ]: Ev2DeflectorTransmission -  HS Short To Power internal";
  gc_ErrTranslation_fr_Text919 : WSTRING(59) := " [PIN_159 ]: Ev2DeflectorTransmission -  HS Short To Ground";
  gc_ErrTranslation_fr_Text920 : WSTRING(62) := " [PIN_159 ]: Ev2DeflectorTransmission -  Internal Driver Error";
  gc_ErrTranslation_fr_Text921 : WSTRING(70) := " [-]: , ,  - Condition erreur correspondante a SPN-  DB Nv Store Error";
  gc_ErrTranslation_fr_Text922 : WSTRING(71) := " [-]: , ,  - Condition erreur correspondante a SPN-  DB Nv Backup Error";
  gc_ErrTranslation_fr_Text923 : WSTRING(70) := " [-]: , ,  - Condition erreur correspondante a SPN-  DB Nv Store Error";
  gc_ErrTranslation_fr_Text924 : WSTRING(71) := " [-]: , ,  - Condition erreur correspondante a SPN-  DB Nv Backup Error";
  gc_ErrTranslation_fr_Text925 : WSTRING(6) := " [-]: ";
  gc_ErrTranslation_fr_Text926 : WSTRING(70) := " [-]: , ,  - Condition erreur correspondante a SPN-  DB Nv Store Error";
  gc_ErrTranslation_fr_Text927 : WSTRING(71) := " [-]: , ,  - Condition erreur correspondante a SPN-  DB Nv Backup Error";
  gc_ErrTranslation_fr_Text928 : WSTRING(6) := " [-]: ";
  gc_ErrTranslation_fr_Text929 : WSTRING(70) := " [-]: , ,  - Condition erreur correspondante a SPN-  DB Nv Store Error";
  gc_ErrTranslation_fr_Text930 : WSTRING(71) := " [-]: , ,  - Condition erreur correspondante a SPN-  DB Nv Backup Error";
  gc_ErrTranslation_fr_Text931 : WSTRING(6) := " [-]: ";
  gc_ErrTranslation_fr_Text932 : WSTRING(70) := " [-]: , ,  - Condition erreur correspondante a SPN-  DB Nv Store Error";
  gc_ErrTranslation_fr_Text933 : WSTRING(71) := " [-]: , ,  - Condition erreur correspondante a SPN-  DB Nv Backup Error";
  gc_ErrTranslation_fr_Text934 : WSTRING(6) := " [-]: ";
  gc_ErrTranslation_fr_Text935 : WSTRING(70) := " [-]: , ,  - Condition erreur correspondante a SPN-  DB Nv Store Error";
  gc_ErrTranslation_fr_Text936 : WSTRING(71) := " [-]: , ,  - Condition erreur correspondante a SPN-  DB Nv Backup Error";
  gc_ErrTranslation_fr_Text937 : WSTRING(6) := " [-]: ";
  gc_ErrTranslation_fr_Text938 : WSTRING(72) := " [PIN_188 ]: SupplyPvgLeftTrack -  HS OpenLoad / Short To Power external";
  gc_ErrTranslation_fr_Text939 : WSTRING(61) := " [PIN_188 ]: SupplyPvgLeftTrack -  HS Short To Power internal";
  gc_ErrTranslation_fr_Text940 : WSTRING(53) := " [PIN_188 ]: SupplyPvgLeftTrack -  HS Short To Ground";
  gc_ErrTranslation_fr_Text941 : WSTRING(56) := " [PIN_188 ]: SupplyPvgLeftTrack -  Internal Driver Error";
  gc_ErrTranslation_fr_Text942 : WSTRING(70) := " [-]: , ,  - Condition erreur correspondante a SPN-  DB Nv Store Error";
  gc_ErrTranslation_fr_Text943 : WSTRING(71) := " [-]: , ,  - Condition erreur correspondante a SPN-  DB Nv Backup Error";
  gc_ErrTranslation_fr_Text944 : WSTRING(6) := " [-]: ";
  gc_ErrTranslation_fr_Text945 : WSTRING(70) := " [-]: , ,  - Condition erreur correspondante a SPN-  DB Nv Store Error";
  gc_ErrTranslation_fr_Text946 : WSTRING(71) := " [-]: , ,  - Condition erreur correspondante a SPN-  DB Nv Backup Error";
  gc_ErrTranslation_fr_Text947 : WSTRING(6) := " [-]: ";
  gc_ErrTranslation_fr_Text948 : WSTRING(26) := "Time out of cyclic message";
  gc_ErrTranslation_fr_Text949 : WSTRING(70) := " [-]: , ,  - Condition erreur correspondante a SPN-  DB Nv Store Error";
  gc_ErrTranslation_fr_Text950 : WSTRING(71) := " [-]: , ,  - Condition erreur correspondante a SPN-  DB Nv Backup Error";
  gc_ErrTranslation_fr_Text951 : WSTRING(6) := " [-]: ";
  gc_ErrTranslation_fr_Text952 : WSTRING(26) := "Time out of cyclic message";
  gc_ErrTranslation_fr_Text953 : WSTRING(48) := " [-]: DeversFrame1 -  Time out of cyclic message";
  gc_ErrTranslation_fr_Text954 : WSTRING(26) := "Time out of cyclic message";
  gc_ErrTranslation_fr_Text955 : WSTRING(26) := "Time out of cyclic message";
  gc_ErrTranslation_fr_Text956 : WSTRING(26) := "Time out of cyclic message";
  gc_ErrTranslation_fr_Text957 : WSTRING(26) := "Time out of cyclic message";
  gc_ErrTranslation_fr_Text958 : WSTRING(26) := "Time out of cyclic message";
  gc_ErrTranslation_fr_Text959 : WSTRING(23) := "Message Buffer Overflow";
  gc_ErrTranslation_fr_Text960 : WSTRING(15) := "Invalid Message";
  gc_ErrTranslation_fr_Text961 : WSTRING(8) := "Timeslot";
  gc_ErrTranslation_fr_Text962 : WSTRING(26) := "Time out of cyclic message";
  gc_ErrTranslation_fr_Text963 : WSTRING(23) := "Message Buffer Overflow";
  gc_ErrTranslation_fr_Text964 : WSTRING(15) := "Invalid Message";
  gc_ErrTranslation_fr_Text965 : WSTRING(8) := "Timeslot";
  gc_ErrTranslation_fr_Text966 : WSTRING(26) := "Time out of cyclic message";
  gc_ErrTranslation_fr_Text967 : WSTRING(23) := "Message Buffer Overflow";
  gc_ErrTranslation_fr_Text968 : WSTRING(15) := "Invalid Message";
  gc_ErrTranslation_fr_Text969 : WSTRING(8) := "Timeslot";
  gc_ErrTranslation_fr_Text970 : WSTRING(26) := "Time out of cyclic message";
  gc_ErrTranslation_fr_Text971 : WSTRING(51) := " [-]: EncodeurTurret1 -  Time out of cyclic message";
  gc_ErrTranslation_fr_Text972 : WSTRING(51) := " [-]: EncodeurTurret2 -  Time out of cyclic message";
  gc_ErrTranslation_fr_Text973 : WSTRING(70) := " [-]: , ,  - Condition erreur correspondante a SPN-  DB Nv Store Error";
  gc_ErrTranslation_fr_Text974 : WSTRING(71) := " [-]: , ,  - Condition erreur correspondante a SPN-  DB Nv Backup Error";
  gc_ErrTranslation_fr_Text975 : WSTRING(57) := " [-]: Msg1C0RcvFromEvision7 -  Time out of cyclic message";
  gc_ErrTranslation_fr_Text976 : WSTRING(6) := " [-]: ";
  gc_ErrTranslation_fr_Text977 : WSTRING(49) := " [-]: DataRcvFromC1 -  Time out of cyclic message";
  gc_ErrTranslation_fr_Text978 : WSTRING(23) := "Message Buffer Overflow";
  gc_ErrTranslation_fr_Text979 : WSTRING(15) := "Invalid Message";
  gc_ErrTranslation_fr_Text980 : WSTRING(8) := "Timeslot";
  gc_ErrTranslation_fr_Text981 : WSTRING(70) := " [-]: , ,  - Condition erreur correspondante a SPN-  DB Nv Store Error";
  gc_ErrTranslation_fr_Text982 : WSTRING(71) := " [-]: , ,  - Condition erreur correspondante a SPN-  DB Nv Backup Error";
  gc_ErrTranslation_fr_Text983 : WSTRING(6) := " [-]: ";
  gc_ErrTranslation_fr_Text984 : WSTRING(69) := " [-]: , ,  - Condition erreur correspondante a SPN-  DM_LIST_OVERFLOW";
  gc_ErrTranslation_fr_Text985 : WSTRING(69) := " [-]: , ,  - Condition erreur correspondante a SPN-  DM_LIST_OVERFLOW";
  gc_ErrTranslation_fr_Text986 : WSTRING(55) := " [-]: SpecificErrorC0 -  Inconsistency selector signals";
  gc_ErrTranslation_fr_Text987 : WSTRING(76) := " [-]: SpecificErrorC0 -  Inconsistency abutment turret track and center size";
  gc_ErrTranslation_fr_Text988 : WSTRING(55) := " [-]: SpecificErrorC0 -  Inconsistency abutment nacelle";
  gc_ErrTranslation_fr_Text989 : WSTRING(80) := " [-]: SpecificErrorC0 -  Inconsistency of pressure and control of solenoid valve";
  gc_ErrTranslation_fr_Text990 : WSTRING(60) := " [-]: SpecificErrorC0 -  control pressure accumulator brakes";
  gc_ErrTranslation_fr_Text991 : WSTRING(65) := " [-]: SpecificErrorC0 -  Hydraulic temperature fault mode crawler";
  gc_ErrTranslation_fr_Text992 : WSTRING(54) := " [-]: SpecificErrorC1 -  Overlaod sensor fault 1 and 2";
  gc_ErrTranslation_fr_Text993 : WSTRING(94) := " [-]: SpecificErrorC1 -  Internal defaut and inconsistency beetween two channels and error can";
  gc_ErrTranslation_fr_Text994 : WSTRING(25) := " [-]: SpecificErrorC1 -  ";
  gc_ErrTranslation_fr_Text995 : WSTRING(36) := " [-]: SpecificErrorC1 -  Input at 1 ";
  gc_ErrTranslation_fr_Text996 : WSTRING(58) := " [-]: SpecificErrorC1 -  Default S1 or S2 pressure sensors";
  gc_ErrTranslation_fr_Text997 : WSTRING(70) := " [-]: , ,  - Condition erreur correspondante a SPN-  DB Nv Store Error";
  gc_ErrTranslation_fr_Text998 : WSTRING(71) := " [-]: , ,  - Condition erreur correspondante a SPN-  DB Nv Backup Error";
  gc_ErrTranslation_fr_Text999 : WSTRING(6) := " [-]: ";
  gc_ErrTranslation_fr_Text1000 : WSTRING(70) := " [-]: , ,  - Condition erreur correspondante a SPN-  DB Nv Store Error";
  gc_ErrTranslation_fr_Text1001 : WSTRING(71) := " [-]: , ,  - Condition erreur correspondante a SPN-  DB Nv Backup Error";
  gc_ErrTranslation_fr_Text1002 : WSTRING(6) := " [-]: ";
  gc_ErrTranslation_fr_Text1003 : WSTRING(70) := " [-]: , ,  - Condition erreur correspondante a SPN-  DB Nv Store Error";
  gc_ErrTranslation_fr_Text1004 : WSTRING(51) := " [-]: TelescopeFrame1 -  Time out of cyclic message";
  gc_ErrTranslation_fr_Text1005 : WSTRING(71) := " [-]: , ,  - Condition erreur correspondante a SPN-  DB Nv Backup Error";
  gc_ErrTranslation_fr_Text1006 : WSTRING(6) := " [-]: ";
  gc_ErrTranslation_fr_Text1007 : WSTRING(51) := " [-]: TelescopeFrame2 -  Time out of cyclic message";
  gc_ErrTranslation_fr_Text1008 : WSTRING(70) := " [-]: , ,  - Condition erreur correspondante a SPN-  DB Nv Store Error";
  gc_ErrTranslation_fr_Text1009 : WSTRING(71) := " [-]: , ,  - Condition erreur correspondante a SPN-  DB Nv Backup Error";
  gc_ErrTranslation_fr_Text1010 : WSTRING(6) := " [-]: ";
  gc_ErrTranslation_fr_Text1011 : WSTRING(52) := " [-]: SendToC1RadioCmd -  Time out of cyclic message";
  gc_ErrTranslation_fr_Text1012 : WSTRING(48) := " [-]: SendToC1RadioCmd - Message Buffer Overflow";
  gc_ErrTranslation_fr_Text1013 : WSTRING(40) := " [-]: SendToC1RadioCmd - Invalid Message";
  gc_ErrTranslation_fr_Text1014 : WSTRING(70) := " [-]: , ,  - Condition erreur correspondante a SPN-  DB Nv Store Error";
  gc_ErrTranslation_fr_Text1015 : WSTRING(33) := " [-]: SendToC1RadioCmd - Timeslot";
  gc_ErrTranslation_fr_Text1016 : WSTRING(23) := "Message Buffer Overflow";
  gc_ErrTranslation_fr_Text1017 : WSTRING(48) := " [-]: DataSendToC1 -  Time out of cyclic message";
  gc_ErrTranslation_fr_Text1018 : WSTRING(15) := "Invalid Message";
  gc_ErrTranslation_fr_Text1019 : WSTRING(71) := " [-]: , ,  - Condition erreur correspondante a SPN-  DB Nv Backup Error";
  gc_ErrTranslation_fr_Text1020 : WSTRING(8) := "Timeslot";
  gc_ErrTranslation_fr_Text1021 : WSTRING(6) := " [-]: ";
  gc_ErrTranslation_fr_Text1022 : WSTRING(26) := "Time out of cyclic message";
  gc_ErrTranslation_fr_Text1023 : WSTRING(70) := " [-]: , ,  - Condition erreur correspondante a SPN-  DB Nv Store Error";
  gc_ErrTranslation_fr_Text1024 : WSTRING(26) := "Time out of cyclic message";
  gc_ErrTranslation_fr_Text1025 : WSTRING(71) := " [-]: , ,  - Condition erreur correspondante a SPN-  DB Nv Backup Error";
  gc_ErrTranslation_fr_Text1026 : WSTRING(6) := " [-]: ";
  gc_ErrTranslation_fr_Text1027 : WSTRING(23) := "Message Buffer Overflow";
  gc_ErrTranslation_fr_Text1028 : WSTRING(26) := "Time out of cyclic message";
  gc_ErrTranslation_fr_Text1029 : WSTRING(15) := "Invalid Message";
  gc_ErrTranslation_fr_Text1030 : WSTRING(8) := "Timeslot";
  gc_ErrTranslation_fr_Text1031 : WSTRING(23) := "Message Buffer Overflow";
  gc_ErrTranslation_fr_Text1032 : WSTRING(26) := "Time out of cyclic message";
  gc_ErrTranslation_fr_Text1033 : WSTRING(15) := "Invalid Message";
  gc_ErrTranslation_fr_Text1034 : WSTRING(8) := "Timeslot";
  gc_ErrTranslation_fr_Text1035 : WSTRING(47) := " [-]: MastMeasure -  Time out of cyclic message";
  gc_ErrTranslation_fr_Text1036 : WSTRING(23) := "Message Buffer Overflow";
  gc_ErrTranslation_fr_Text1037 : WSTRING(49) := " [-]: Data2SendToC1 -  Time out of cyclic message";
  gc_ErrTranslation_fr_Text1038 : WSTRING(15) := "Invalid Message";
  gc_ErrTranslation_fr_Text1039 : WSTRING(8) := "Timeslot";
  gc_ErrTranslation_fr_Text1040 : WSTRING(23) := "Message Buffer Overflow";
  gc_ErrTranslation_fr_Text1041 : WSTRING(50) := " [-]: Data2RdvFromC1 -  Time out of cyclic message";
  gc_ErrTranslation_fr_Text1042 : WSTRING(15) := "Invalid Message";
  gc_ErrTranslation_fr_Text1043 : WSTRING(8) := "Timeslot";
  gc_ErrTranslation_fr_Text1044 : WSTRING(57) := " [-]: Msg1C0RcvFromEvision7 -  Time out of cyclic message";
  gc_ErrTranslation_fr_Text1045 : WSTRING(70) := " [-]: , ,  - Condition erreur correspondante a SPN-  DB Nv Store Error";
  gc_ErrTranslation_fr_Text1046 : WSTRING(71) := " [-]: , ,  - Condition erreur correspondante a SPN-  DB Nv Backup Error";
  gc_ErrTranslation_fr_Text1047 : WSTRING(6) := " [-]: ";
  gc_ErrTranslation_fr_Text1048 : WSTRING(70) := " [-]: , ,  - Condition erreur correspondante a SPN-  DB Nv Store Error";
  gc_ErrTranslation_fr_Text1049 : WSTRING(71) := " [-]: , ,  - Condition erreur correspondante a SPN-  DB Nv Backup Error";
  gc_ErrTranslation_fr_Text1050 : WSTRING(6) := " [-]: ";
  gc_ErrTranslation_fr_Text1051 : WSTRING(70) := " [-]: , ,  - Condition erreur correspondante a SPN-  DB Nv Store Error";
  gc_ErrTranslation_fr_Text1052 : WSTRING(71) := " [-]: , ,  - Condition erreur correspondante a SPN-  DB Nv Backup Error";
  gc_ErrTranslation_fr_Text1053 : WSTRING(6) := " [-]: ";
  gc_ErrTranslation_fr_Text1054 : WSTRING(23) := "Message Buffer Overflow";
  gc_ErrTranslation_fr_Text1055 : WSTRING(49) := " [-]: Data3SendToC1 -  Time out of cyclic message";
  gc_ErrTranslation_fr_Text1056 : WSTRING(15) := "Invalid Message";
  gc_ErrTranslation_fr_Text1057 : WSTRING(8) := "Timeslot";
  gc_ErrTranslation_fr_Text1058 : WSTRING(26) := "Time out of cyclic message";
  gc_ErrTranslation_fr_Text1059 : WSTRING(70) := " [-]: , ,  - Condition erreur correspondante a SPN-  DB Nv Store Error";
  gc_ErrTranslation_fr_Text1060 : WSTRING(71) := " [-]: , ,  - Condition erreur correspondante a SPN-  DB Nv Backup Error";
  gc_ErrTranslation_fr_Text1061 : WSTRING(6) := " [-]: ";
  gc_ErrTranslation_fr_Text1062 : WSTRING(26) := "Time out of cyclic message";
  gc_ErrTranslation_fr_Text1063 : WSTRING(26) := "Time out of cyclic message";
  gc_ErrTranslation_fr_Text1064 : WSTRING(23) := "Message Buffer Overflow";
  gc_ErrTranslation_fr_Text1065 : WSTRING(26) := "Time out of cyclic message";
  gc_ErrTranslation_fr_Text1066 : WSTRING(15) := "Invalid Message";
  gc_ErrTranslation_fr_Text1067 : WSTRING(8) := "Timeslot";
  gc_ErrTranslation_fr_Text1068 : WSTRING(23) := "Message Buffer Overflow";
  gc_ErrTranslation_fr_Text1069 : WSTRING(50) := " [-]: Data3RcvFromC1 -  Time out of cyclic message";
  gc_ErrTranslation_fr_Text1070 : WSTRING(15) := "Invalid Message";
  gc_ErrTranslation_fr_Text1071 : WSTRING(8) := "Timeslot";
  gc_ErrTranslation_fr_Text1072 : WSTRING(47) := " [-]: SpecificErrorC1_3 -  Overlaod is detected";
  gc_ErrTranslation_fr_Text1073 : WSTRING(64) := " [-]: SpecificErrorC1_3 -  Failt of Ev park brake axle oscillant";
  gc_ErrTranslation_fr_Text1074 : WSTRING(59) := " [-]: SpecificErrorC1_3 -  Fault of Ev park brake axle fixe";
  gc_ErrTranslation_fr_Text1075 : WSTRING(67) := " [-]: SpecificErrorC1_3 -  Fault of Ev service brake axle oscillant";
  gc_ErrTranslation_fr_Text1076 : WSTRING(62) := " [-]: SpecificErrorC1_3 -  Fault of Ev service brake axle fixe";
  gc_ErrTranslation_fr_Text1077 : WSTRING(60) := " [-]: SpecificErrorC0_3 -  Coherence pilotage PVG track left";
  gc_ErrTranslation_fr_Text1078 : WSTRING(77) := " [-]: SpecificErrorC0_4 -  Number of cycle brake perform is over at threshold";
  gc_ErrTranslation_fr_Text1079 : WSTRING(96) := " [-]: SpecificErrorC0_4 -  Test brakes not validated , exceeded critical number of brake perform";
  gc_ErrTranslation_fr_Text1080 : WSTRING(58) := " [-]: SpecificErrorC0_4 -  Check coherence option of light";
  gc_ErrTranslation_fr_Text1081 : WSTRING(65) := " [-]: SpecificErrorC0_4 -  Right basket sensor inconsistency NcNo";
  gc_ErrTranslation_fr_Text1082 : WSTRING(64) := " [-]: SpecificErrorC0_2 -  Hydraulic temperature fault mode rail";
  gc_ErrTranslation_fr_Text1083 : WSTRING(68) := " [-]: SpecificErrorC0_2 -  Hydraulic temperature alarme mode crawler";
  gc_ErrTranslation_fr_Text1084 : WSTRING(68) := " [-]: SpecificErrorC0_2 -  Hydraulic temperature alarme mode crawler";
  gc_ErrTranslation_fr_Text1085 : WSTRING(89) := " [-]: SpecificErrorC0_2 -  Inconsistency beetween high and low position of axle oscillant";
  gc_ErrTranslation_fr_Text1086 : WSTRING(84) := " [-]: SpecificErrorC0_2 -  Inconsistency beetween high and low position of axle fixe";
  gc_ErrTranslation_fr_Text1087 : WSTRING(69) := " [-]: SpecificErrorC0_2 -  both sensors do not show consistent values";
  gc_ErrTranslation_fr_Text1088 : WSTRING(69) := " [-]: SpecificErrorC0_2 -  both sensors do not show consistent values";
  gc_ErrTranslation_fr_Text1089 : WSTRING(63) := " [-]: SpecificErrorC0_2 -  exceeding the PV overspeed threshold";
  gc_ErrTranslation_fr_Text1090 : WSTRING(63) := " [-]: SpecificErrorC0_3 -  exceeding the GV overspeed threshold";
  gc_ErrTranslation_fr_Text1091 : WSTRING(101) := " [-]: SpecificErrorC0_3 -  CAN communication problem, inconsistency with option, Inconsistent measure";
  gc_ErrTranslation_fr_Text1092 : WSTRING(27) := " [-]: SpecificErrorC0_3 -  ";
  gc_ErrTranslation_fr_Text1093 : WSTRING(27) := " [-]: SpecificErrorC0_3 -  ";
  gc_ErrTranslation_fr_Text1094 : WSTRING(80) := " [-]: SpecificErrorC0_3 -  Inconsistency check position foled of delta and arrow";
  gc_ErrTranslation_fr_Text1095 : WSTRING(74) := " [-]: SpecificErrorC0_3 -  Inconsistency boths 2 channels or can faillures";
  gc_ErrTranslation_fr_Text1096 : WSTRING(27) := " [-]: SpecificErrorC0_3 -  ";
  gc_ErrTranslation_fr_Text1097 : WSTRING(61) := " [-]: SpecificErrorC0_4 -  Coherence pilotage PVG track right";
  gc_ErrTranslation_fr_Text1098 : WSTRING(64) := " [-]: SpecificErrorC0_4 -  Left basket sensor inconsistency NcNo";
  gc_ErrTranslation_fr_Text1099 : WSTRING(78) := " [-]: SpecificErrorC0_4 -  Inconsistency beetween left and right basket sensor";
  gc_ErrTranslation_fr_Text1100 : WSTRING(38) := " [-]: SpecificErrorC0_4 -  Active Help";
  gc_ErrTranslation_fr_Text1101 : WSTRING(27) := " [-]: SpecificErrorC1_3 -  ";
  gc_ErrTranslation_fr_Text1102 : WSTRING(54) := " [-]: FAiluresC1SendToC0 -  Time out of cyclic message";
  gc_ErrTranslation_fr_Text1103 : WSTRING(48) := " [-]: DeversFrame2 -  Time out of cyclic message";
  gc_ErrTranslation_fr_Text1104 : WSTRING(80) := " [-]: SpecificErrorC1_3 -  Inconsistency check position foled of delta and arrow";
  gc_ErrTranslation_fr_Text1105 : WSTRING(66) := " [-]: SpecificErrorC1_3 -  Inconsistency check of telescope sensor";
  gc_ErrTranslation_fr_Text1106 : WSTRING(23) := "Message Buffer Overflow";
  gc_ErrTranslation_fr_Text1107 : WSTRING(15) := "Invalid Message";
  gc_ErrTranslation_fr_Text1108 : WSTRING(8) := "Timeslot";
  gc_ErrTranslation_fr_Text1109 : WSTRING(54) := " [-]: FailuresC0SendToC1 -  Time out of cyclic message";
  gc_ErrTranslation_fr_Text1110 : WSTRING(23) := "Message Buffer Overflow";
  gc_ErrTranslation_fr_Text1111 : WSTRING(15) := "Invalid Message";
  gc_ErrTranslation_fr_Text1112 : WSTRING(8) := "Timeslot";
  gc_ErrTranslation_fr_Text1113 : WSTRING(51) := " [-]: Msg1RcvFromOpus -  Time out of cyclic message";
  gc_ErrTranslation_fr_Text1114 : WSTRING(51) := " [-]: Msg1RcvFromOpus -  Time out of cyclic message";
  gc_ErrTranslation_fr_Text1115 : WSTRING(51) := " [-]: Data4C0SendToC1 -  Time out of cyclic message";
  gc_ErrTranslation_fr_Text1116 : WSTRING(51) := " [-]: Data4C1SendToC0 -  Time out of cyclic message";
  gc_ErrTranslation_fr_Text1117 : WSTRING(23) := "Message Buffer Overflow";
  gc_ErrTranslation_fr_Text1118 : WSTRING(15) := "Invalid Message";
  gc_ErrTranslation_fr_Text1119 : WSTRING(8) := "Timeslot";
  gc_ErrTranslation_fr_Text1120 : WSTRING(23) := "Message Buffer Overflow";
  gc_ErrTranslation_fr_Text1121 : WSTRING(15) := "Invalid Message";
  gc_ErrTranslation_fr_Text1122 : WSTRING(8) := "Timeslot";
  gc_ErrTranslation_fr_Text1123 : WSTRING(26) := "Time out of cyclic message";
  gc_ErrTranslation_fr_Text1124 : WSTRING(26) := "Time out of cyclic message";
  gc_ErrTranslation_fr_Text1125 : WSTRING(82) := " [-]: SpecificErrorC1_4 -  Overloadd detected on motor default light ouput of 48XS";
  gc_ErrTranslation_fr_Text1126 : WSTRING(81) := " [-]: SpecificErrorC1_4 -  Openload detected on motor default light ouput of 48XS";
  gc_ErrTranslation_fr_Text1127 : WSTRING(77) := " [-]: SpecificErrorC1_4 -  Overload detected on overlaod light output of 48xs";
  gc_ErrTranslation_fr_Text1128 : WSTRING(77) := " [-]: SpecificErrorC1_4 -  Openload detected on overload light output of 48xs";
  gc_ErrTranslation_fr_Text1129 : WSTRING(68) := " [-]: SpecificErrorC1_4 -  Overload detected on buzzer ouput of 48xs";
  gc_ErrTranslation_fr_Text1130 : WSTRING(69) := " [-]: SpecificErrorC1_4 -  Openload detected on buzzer output of 48xs";
  gc_ErrTranslation_fr_Text1131 : WSTRING(76) := " [-]: SpecificErrorC1_4 -  Overlaod detected on warming light output of 48xs";
  gc_ErrTranslation_fr_Text1132 : WSTRING(76) := " [-]: SpecificErrorC1_4 -  Opendload detected on warming light ouput of 48xs";
  gc_ErrTranslation_fr_Text1133 : WSTRING(83) := " [-]: SpecificErrorC1_5 -  Overlaod detected on devers default light output of 48xs";
  gc_ErrTranslation_fr_Text1134 : WSTRING(83) := " [-]: SpecificErrorC1_5 -  Openload detected on devers default light output of 48xs";
  gc_ErrTranslation_fr_Text1135 : WSTRING(69) := " [-]: SpecificErrorC1_5 -  Overlaod detected on gas oil light of 4x8s";
  gc_ErrTranslation_fr_Text1136 : WSTRING(69) := " [-]: SpecificErrorC1_5 -  Openload detected on gas oil light of 48xs";
  gc_ErrTranslation_fr_Text1137 : WSTRING(68) := " [-]: SpecificErrorC1_5 -  Overload detected on white lights of 48xs";
  gc_ErrTranslation_fr_Text1138 : WSTRING(68) := " [-]: SpecificErrorC1_5 -  Openload detected on white lights of 48xs";
  gc_ErrTranslation_fr_Text1139 : WSTRING(72) := " [-]: SpecificErrorC1_5 -  Overload detected on red lights ouput of 48xs";
  gc_ErrTranslation_fr_Text1140 : WSTRING(73) := " [-]: SpecificErrorC1_5 -  Openload detected on red lights output of 48xs";
  gc_ErrTranslation_fr_Text1141 : WSTRING(82) := " [-]: SpecificErrorC0_6 -  Overloadd detected on motor default light ouput of 48XS";
  gc_ErrTranslation_fr_Text1142 : WSTRING(81) := " [-]: SpecificErrorC0_6 -  Openload detected on motor default light ouput of 48XS";
  gc_ErrTranslation_fr_Text1143 : WSTRING(77) := " [-]: SpecificErrorC0_6 -  Overload detected on overlaod light output of 48xs";
  gc_ErrTranslation_fr_Text1144 : WSTRING(77) := " [-]: SpecificErrorC0_6 -  Overload detected on overlaod light output of 48xs";
  gc_ErrTranslation_fr_Text1145 : WSTRING(68) := " [-]: SpecificErrorC0_6 -  Overload detected on buzzer ouput of 48xs";
  gc_ErrTranslation_fr_Text1146 : WSTRING(68) := " [-]: SpecificErrorC0_6 -  Overload detected on buzzer ouput of 48xs";
  gc_ErrTranslation_fr_Text1147 : WSTRING(76) := " [-]: SpecificErrorC0_6 -  Overlaod detected on warming light output of 48xs";
  gc_ErrTranslation_fr_Text1148 : WSTRING(76) := " [-]: SpecificErrorC0_6 -  Opendload detected on warming light ouput of 48xs";
  gc_ErrTranslation_fr_Text1149 : WSTRING(83) := " [-]: SpecificErrorC0_7 -  Overlaod detected on devers default light output of 48xs";
  gc_ErrTranslation_fr_Text1150 : WSTRING(83) := " [-]: SpecificErrorC0_7 -  Openload detected on devers default light output of 48xs";
  gc_ErrTranslation_fr_Text1151 : WSTRING(83) := " [-]: SpecificErrorC0_7 -  Openload detected on devers default light output of 48xs";
  gc_ErrTranslation_fr_Text1152 : WSTRING(83) := " [-]: SpecificErrorC0_7 -  Openload detected on devers default light output of 48xs";
  gc_ErrTranslation_fr_Text1153 : WSTRING(68) := " [-]: SpecificErrorC0_7 -  Overload detected on white lights of 48xs";
  gc_ErrTranslation_fr_Text1154 : WSTRING(68) := " [-]: SpecificErrorC0_7 -  Openload detected on white lights of 48xs";
  gc_ErrTranslation_fr_Text1155 : WSTRING(72) := " [-]: SpecificErrorC0_7 -  Overload detected on red lights ouput of 48xs";
  gc_ErrTranslation_fr_Text1156 : WSTRING(73) := " [-]: SpecificErrorC0_7 -  Openload detected on red lights output of 48xs";
  gc_ErrTranslation_fr_Text1157 : WSTRING(44) := "Overload detected on white light ARD of 48xs";
  gc_ErrTranslation_fr_Text1158 : WSTRING(44) := "Openload detected on white light ARD of 48xs";
  gc_ErrTranslation_fr_Text1159 : WSTRING(48) := "Overload detected on red light ARD ouput of 48xs";
  gc_ErrTranslation_fr_Text1160 : WSTRING(44) := "Overload detected on white light ARD of 48xs";
  gc_ErrTranslation_fr_Text1161 : WSTRING(44) := "Openload detected on white light ARD of 48xs";
  gc_ErrTranslation_fr_Text1162 : WSTRING(48) := "Overload detected on red light ARD ouput of 48xs";
  gc_ErrTranslation_fr_Text1163 : WSTRING(49) := "Openload detected on red light ARD output of 48xs";
  gc_ErrTranslation_fr_Text1164 : WSTRING(46) := "Overload detected on white light ar 15746 48XS";
  gc_ErrTranslation_fr_Text1165 : WSTRING(66) := " [-]: SpecificErrorC0_8 -  Out of range joystick delta arm of 48XS";
  gc_ErrTranslation_fr_Text1166 : WSTRING(66) := " [-]: SpecificErrorC0_8 -  Out of range joystick arrow arm of 48XS";
  gc_ErrTranslation_fr_Text1167 : WSTRING(70) := " [-]: SpecificErrorC0_8 -  Out of range joystick telescope arm of 48XS";
  gc_ErrTranslation_fr_Text1168 : WSTRING(72) := " [-]: SpecificErrorC0_8 -  Out of range joystick rotation turret of 48XS";
  gc_ErrTranslation_fr_Text1169 : WSTRING(68) := " [-]: SpecificErrorC0_8 -  Out of range joystick advancement of 48XS";
  gc_ErrTranslation_fr_Text1170 : WSTRING(66) := " [-]: SpecificErrorC1_6 -  Out of range joystick delta arm of 48XS";
  gc_ErrTranslation_fr_Text1171 : WSTRING(66) := " [-]: SpecificErrorC1_6 -  Out of range joystick arrow arm of 48XS";
  gc_ErrTranslation_fr_Text1172 : WSTRING(70) := " [-]: SpecificErrorC1_6 -  Out of range joystick telescope arm of 48XS";
  gc_ErrTranslation_fr_Text1173 : WSTRING(72) := " [-]: SpecificErrorC1_6 -  Out of range joystick rotation turret of 48XS";
  gc_ErrTranslation_fr_Text1174 : WSTRING(68) := " [-]: SpecificErrorC1_6 -  Out of range joystick advancement of 48XS";
  gc_ErrTranslation_fr_Text1175 : WSTRING(46) := "Openload detected on white light ar 15746 48XS";
  gc_ErrTranslation_fr_Text1176 : WSTRING(66) := " [-]: SpecificErrorC1_7 -  HeatBeat State of 48XS  different at OK";
  gc_ErrTranslation_fr_Text1177 : WSTRING(57) := " [-]: SpecificErrorC1_7 - Rm com can radio detected by C0";
  gc_ErrTranslation_fr_Text1178 : WSTRING(26) := "Time out of cyclic message";
  gc_ErrTranslation_fr_Text1179 : WSTRING(26) := "Time out of cyclic message";
  gc_ErrTranslation_fr_Text1180 : WSTRING(0) := "";
  gc_ErrTranslation_fr_Text1181 : WSTRING(0) := "";
  gc_ErrTranslation_fr_Text1182 : WSTRING(0) := "";
  gc_ErrTranslation_fr_Text1183 : WSTRING(0) := "";
  gc_ErrTranslation_fr_Text1184 : WSTRING(0) := "";
  gc_ErrTranslation_fr_Text1185 : WSTRING(0) := "";
  gc_ErrTranslation_fr_Text1186 : WSTRING(0) := "";
  gc_ErrTranslation_fr_Text1187 : WSTRING(0) := "";
  gc_ErrTranslation_fr_Text1188 : WSTRING(0) := "";
  gc_ErrTranslation_fr_Text1189 : WSTRING(0) := "";
  gc_ErrTranslation_fr_Text1190 : WSTRING(0) := "";
  gc_ErrTranslation_fr_Text1191 : WSTRING(0) := "";
  gc_ErrTranslation_fr_Text1192 : WSTRING(0) := "";
  gc_ErrTranslation_fr_Text1193 : WSTRING(0) := "";
